// TIA Portal V16 export
// export: Created 2021-07-12T14:47:18.3595823Z, ExportSetting WithDefaults, DisplayName Totally Integrated Automation Portal, DisplayVersion V16, DisplayName TIA Portal Version Control Interface, DisplayVersion V16, DisplayName TIA Portal Openness, DisplayVersion V16, DisplayName STEP 7 Professional, DisplayVersion V16, DisplayName STEP 7 Safety, DisplayVersion V16, DisplayName WinCC Professional, DisplayVersion V16
TYPE "LSimaHydTO_typeStatusVChar"
TITLE = LSimaHydTO_typeStatusVChar
// Indicates the status of valve characteristic data
// stored: IsFailsafeCompliant false
   STRUCT
      ActualVChar : UInt := 0;   // Currently effective valve characteristic DB number
   END_STRUCT;
END_TYPE
